(* IEC 61131-3 sources: windowtracking/src/EventHandler, 13 files *)

(* ---- EventStatus.st ---- *)
NAMESPACE Simatic.Ax.WindowTracking.EventHandler

    TYPE
        EventStatus : (Undefined, Finished, Error, NullReference, NotEnabled) := Undefined;
    END_TYPE

END_NAMESPACE

(* ---- IExit.st ---- *)
NAMESPACE Simatic.Ax.WindowTracking.Exits
    INTERFACE IExit
        METHOD IsReady : BOOL
        END_METHOD
    END_INTERFACE
END_NAMESPACE

(* ---- IExitPoint.st ---- *)
NAMESPACE Simatic.Ax.WindowTracking.EventHandler
    INTERFACE IExitPoint
        METHOD IsReady : BOOL
        END_METHOD
    END_INTERFACE
END_NAMESPACE

(* ---- ISortDecission.st ---- *)
USING Simatic.Ax.WindowTracking.EventHandler;
USING Simatic.Ax.WindowTracking.Trigger;
NAMESPACE Simatic.Ax.WindowTracking
    INTERFACE ISortDecission
        METHOD Check : BOOL
            VAR_INPUT
                tw : ITransportWindow;
                te : IVirtualTrigger;
                exitpoint : IExitPoint;
            END_VAR
        END_METHOD
    END_INTERFACE
END_NAMESPACE

(* ---- ITriggerEvent.st ---- *)
USING Simatic.Ax.WindowTracking.Trigger;

NAMESPACE Simatic.Ax.WindowTracking.EventHandler
    INTERFACE ITriggerEvent
        METHOD Action : EventStatus
            VAR_INPUT
                te : IVirtualTrigger;
                tw : ITransportWindow;
            END_VAR
        END_METHOD
    END_INTERFACE

END_NAMESPACE

(* ---- IUserDefinedEvent.st ---- *)
NAMESPACE Simatic.Ax.WindowTracking
    INTERFACE IUserDefinedEvent
        METHOD Action : EventStatus
            VAR_INPUT
                te : IVirtualTrigger;
                tw : ITransportWindow;
            END_VAR
        END_METHOD
    END_INTERFACE

END_NAMESPACE

(* ---- ClearWindow.st ---- *)
USING Simatic.Ax.WindowTracking.Events;
USING Simatic.Ax.WindowTracking.Trigger;
NAMESPACE Simatic.Ax.WindowTracking.EventHandler
    CLASS ClearWindow IMPLEMENTS ITriggerEvent
        VAR PUBLIC
            WindowList : ITransportWindowsCleanup;
        END_VAR

        METHOD PUBLIC Action : EventStatus
            VAR_INPUT
                te : IVirtualTrigger;
                tw : ITransportWindow;
            END_VAR
            // Remove oldest window from list
            WindowList.Remove();
            ;
        END_METHOD
    END_CLASS
END_NAMESPACE

(* ---- ClearWindowEvent.st ---- *)
USING Simatic.Ax.WindowTracking.Trigger;

NAMESPACE Simatic.Ax.WindowTracking.EventHandler
    CLASS ClearWindowEvent IMPLEMENTS ITriggerEvent
        VAR PUBLIC
            WindowList : ITransportWindowsCleanup;
        END_VAR

        METHOD PUBLIC Action : EventStatus
            VAR_INPUT
                te : IVirtualTrigger;
                tw : ITransportWindow;
            END_VAR
            // Remove oldest window from list
            WindowList.Remove();
            ;
        END_METHOD
    END_CLASS
END_NAMESPACE

(* ---- ExitPoint.st ---- *)
USING Simatic.Ax.WindowTracking.Events;
USING Simatic.Ax.WindowTracking.Trigger;

NAMESPACE Simatic.Ax.WindowTracking.EventHandler
    CLASS ExitPoint IMPLEMENTS ITriggerEvent, IExitPoint

        VAR PUBLIC
            SortDecission : ISortDecission;
        END_VAR

        METHOD PUBLIC Action : EventStatus
            VAR_INPUT
                te : IVirtualTrigger;
                tw : ITransportWindow;
            END_VAR
            VAR_TEMP
                _sortItem : BOOL;
            END_VAR
            _sortItem := SortDecission.Check(tw := tw, te := te, exitpoint := THIS);

        END_METHOD

        METHOD PUBLIC IsReady : BOOL
            IsReady := TRUE;
        END_METHOD
    END_CLASS
END_NAMESPACE

(* ---- SortDecisionEvent.st ---- *)
NAMESPACE Simatic.Ax.WindowTracking
    CLASS SortDecisionEvent IMPLEMENTS ITriggerEvent

        VAR PUBLIC
            SortStrategy : ISortStrategy;
            ExitHandler : IExitPointHandler;
            EventBefore : IUserDefinedEvent;
            EventAfter : IUserDefinedEvent;
        END_VAR

        METHOD PUBLIC Action : EventStatus
            VAR_INPUT
                te : IVirtualTrigger;
                tw : ITransportWindow;
            END_VAR
            VAR_TEMP
                _check : BOOL;
            END_VAR

            IF (SortStrategy = NULL) THEN
                Action := EventStatus#NullReference;
                RETURN;
            END_IF;
            IF (ExitHandler = NULL) THEN
                Action := EventStatus#NullReference;
                RETURN;
            END_IF;

            _check := SortStrategy.Check(tw := tw, te := te, exitpoint := ExitHandler);

            IF (_check) THEN
                // Activate additional user defined event before
                IF (EventBefore <> NULL) THEN
                    EventBefore.Action(tw := tw, te := te);
                END_IF;

                ExitHandler.Activate();
                Action := EventStatus#Finished;

                // Activate additional user defined event after
                IF (EventAfter <> NULL) THEN
                    EventAfter.Action(tw := tw, te := te);
                END_IF;

                RETURN;
            END_IF;

            Action := EventStatus#Undefined;

        END_METHOD

        METHOD PUBLIC ActionAfter : EventStatus
            VAR_INPUT
                te : IVirtualTrigger;
                tw : ITransportWindow;
            END_VAR
            ; // do nothing
        END_METHOD
    END_CLASS
END_NAMESPACE

(* ---- SortDecissionEvent.st ---- *)
USING Simatic.Ax.WindowTracking.EventHandler;
USING Simatic.Ax.WindowTracking.Trigger;
USING Simatic.Ax.WindowTracking.SortDecission;

NAMESPACE Simatic.Ax.WindowTracking.EventHandler
    CLASS SortDecissionEvent IMPLEMENTS ITriggerEvent

        VAR PUBLIC
            SortDecission : ISortDecission;
            ExitHandler : IExitPointHandler;
        END_VAR

        METHOD PUBLIC Action : EventStatus
            VAR_INPUT
                te : IVirtualTrigger;
                tw : ITransportWindow;
            END_VAR
            VAR_TEMP
                _check : BOOL;
            END_VAR

            IF (SortDecission = NULL) THEN
                Action := EventStatus#NullReference;
                RETURN;
            END_IF;
            IF (ExitHandler = NULL) THEN
                Action := EventStatus#NullReference;
                RETURN;
            END_IF;

            _check := SortDecission.Check(tw := tw, te := te, exitpoint := ExitHandler);

            IF (_check) THEN
                ExitHandler.Activate();
                Action := EventStatus#Finished;
                RETURN;
            END_IF;

            Action := EventStatus#Undefined;

        END_METHOD

    END_CLASS
END_NAMESPACE

(* ---- SortDecissionOneDestination.st ---- *)
USING Simatic.Ax.WindowTracking.Exits;
USING Simatic.Ax.WindowTracking.Trigger;

NAMESPACE Simatic.Ax.WindowTracking.EventHandler
    CLASS SortDecissionOneDestination IMPLEMENTS ISortDecission
        VAR PUBLIC

        END_VAR
        VAR PROTECTED

        END_VAR

        METHOD PUBLIC Check : BOOL
            VAR_INPUT
                o : ITransportWindow;
            END_VAR

            VAR_TEMP
                i : UINT;
                _tp : IVirtualTrigger;
                _exit : IExit;
            END_VAR
            ;
            // Check the destination. Only one Destination is valid!
            // IF (o.GetTriggerPointCount() = UINT#1) THEN
            //     _tp := o.GetTriggerPoint(UINT#0);
            //     // _exit := o.GetExit();

            //     IF (NOT(_tp.IsEnabled())) THEN
            //         Check := FALSE;
            //         RETURN;
            //     END_IF;

            //     IF (NOT(_exit.IsReady())) THEN
            //         Check := FALSE;
            //         RETURN;
            //     END_IF;

            //     Check := TRUE;

            // END_IF;
        END_METHOD
    END_CLASS
END_NAMESPACE

(* ---- TerminateWindowEvent.st ---- *)
NAMESPACE Simatic.Ax.WindowTracking
    CLASS FINAL TerminateWindowEvent IMPLEMENTS ITriggerEvent
        VAR PUBLIC
            WindowList : ITransportWindowsTerminate;
            EventBefore : IUserDefinedEvent;
            EventAfter : IUserDefinedEvent;
        END_VAR

        METHOD PUBLIC Action : EventStatus
            VAR_INPUT
                te : IVirtualTrigger;
                tw : ITransportWindow;
            END_VAR
            ;
        END_METHOD

        METHOD PUBLIC ActionAfter : EventStatus
            VAR_INPUT
                te : IVirtualTrigger;
                tw : ITransportWindow;
            END_VAR
            // Activate additional user defined event before
            IF (EventBefore <> NULL) THEN
                EventBefore.Action(tw := tw, te := te);
            END_IF;

            // Remove oldest window from list
            WindowList.Terminate();

            // Activate additional user defined event after
            IF (EventAfter <> NULL) THEN
                EventAfter.Action(tw := tw, te := te);
            END_IF;
            ;
        END_METHOD
    END_CLASS
END_NAMESPACE
